{attribute 'linkalways'} 
{attribute 'no_explicit_call' := 'This FB is a CLASS and must be accessed using methods or properties'}
{attribute 'enable_dynamic_creation'}
FUNCTION_BLOCK _ETcVnColorTrainingMethod EXTENDS EnumDatatypeBase
VAR
	localData : ETcVnColorTrainingMethod;
	activeData : REFERENCE TO ETcVnColorTrainingMethod;
	enumBaseDatatype : _DINT(localData);
END_VAR

METHOD PRIVATE AddLocalEnumeration
VAR_INPUT
	Enumeration : T_MAXSTRING;
	Value : ETcVnColorTrainingMethod;
END_VAR
AddEnumeration(Enumeration, Value);
END_METHOD

PROPERTY PUBLIC Address : PVOID
GET
Address := ADR(activeData);
END_GET
END_PROPERTY

METHOD PUBLIC ClearReference
VAR_INPUT
END_VAR
activeData REF= localData;
SetBaseDatatypeReference();
END_METHOD

METHOD PUBLIC Clone : I_Datatype
VAR
    pClone : POINTER TO _ETcVnColorTrainingMethod;
END_VAR
pClone := __NEW(_ETcVnColorTrainingMethod(InitialValue := Value));
Clone := pClone^;
END_METHOD

METHOD FB_init : BOOL
VAR_INPUT
	bInitRetains : BOOL; // if TRUE, the retain variables are initialized (warm start / cold start)
	bInCopyCode : BOOL;  // if TRUE, the instance afterwards gets moved into the copy code (online change)
	InitialValue : ETcVnColorTrainingMethod;
END_VAR
localData := InitialValue;
AddBaseDatatype(enumBaseDatatype);
ClearReference();

AddLocalEnumeration('TCVN_CTM_LAB', ETcVnColorTrainingMethod.TCVN_CTM_LAB);
AddLocalEnumeration('TCVN_CTM_RGB', ETcVnColorTrainingMethod.TCVN_CTM_RGB);
END_METHOD

PROPERTY PUBLIC Identifier : T_MAXSTRING
GET
Identifier := 'ETcVnColorTrainingMethod';
END_GET
END_PROPERTY

METHOD IsEnumeratorValueEqual : BOOL
VAR_INPUT
	Enumerator : I_KeyValueForwardEnumerator;
END_VAR
VAR
	storedValue : ETcVnColorTrainingMethod;
END_VAR
IF NOT Enumerator.TryGet(storedValue) THEN
	RETURN;
END_IF

IsEnumeratorValueEqual := storedValue = activeData;
END_METHOD

METHOD PUBLIC MakeReferenceTo
VAR_INPUT
	ReferenceTarget : REFERENCE TO ETcVnColorTrainingMethod;
END_VAR
activeData REF= ReferenceTarget;
SetBaseDatatypeReference();
END_METHOD

METHOD PROTECTED SetBaseDatatypeReference
VAR_INPUT
END_VAR
enumBaseDatatype.MakeReferenceTo(activeData);
END_METHOD

PROPERTY PUBLIC Size : UDINT
GET
Size := SIZEOF(activeData);
END_GET
END_PROPERTY

METHOD TryMakeReferenceTo : BOOL
VAR_INPUT
	Target : I_Datatype;
END_VAR
VAR
	targetAsEnum : I_EnumDatatype;
	pTargetData : POINTER TO ETcVnColorTrainingMethod;
END_VAR
IF NOT Target.TryResolveAsEnumDatatype(targetAsEnum) THEN
	RETURN;
END_IF

IF targetAsEnum.Identifier <> Identifier THEN
	RETURN;
END_IF

pTargetData := Target.Address;
activeData REF= pTargetData^;
SetBaseDatatypeReference();
TryMakeReferenceTo := TRUE;
END_METHOD

PROPERTY PUBLIC Value : ETcVnColorTrainingMethod
GET
Value := activeData;
END_GET
SET
activeData := Value;
END_SET
END_PROPERTY

END_FUNCTION_BLOCK

(* stored: Version 1.1.0.1, ProductVersion 3.1.4024.12
   POU _ETcVnColorTrainingMethod: Id {6028da55-d8a0-0f8d-2afc-d94080e8e5ba}, SpecialFunc None
   Folder Constructor: Id {1bb38a8e-b814-0d41-3d43-d2efa85f6946}
   Folder Private: Id {cf11808f-3c76-0852-2ed6-f98f4ad7fced}
   Folder Protected: Id {f1175831-533e-03d6-3c3a-4faefcf5d79d}
   Method AddLocalEnumeration: Id {b7e3e48d-8aae-04b2-3d6c-7a977cbc5a40}
   Property Address: Id {b6820bd9-1f14-069c-2263-f363a84e71b0}
   Get Get: Id {9ad705a9-391b-01d9-0a6a-2dcb629bfc1d}
   Method ClearReference: Id {638f89f2-5d18-07f7-0871-123cb68304e9}
   Method Clone: Id {82db6a33-a5e5-01a1-14b1-9dd96bf7d688}
   Method FB_init: Id {3580fadd-f501-0afa-1fda-3530e26eb045}
   Property Identifier: Id {0f149496-b3d1-08c6-1eee-49ef345cf84e}
   Get Get: Id {7e3af238-043c-06ad-3e48-49416720f0da}
   Method IsEnumeratorValueEqual: Id {5e1dd4e3-1066-0fbe-2fc3-9e81e510c494}
   Method MakeReferenceTo: Id {ec6f9e4f-cdab-0f8f-384f-b11715e64901}
   Method SetBaseDatatypeReference: Id {766004f2-24a4-08f3-31b6-3a9b0f3660dd}
   Property Size: Id {9274ffc8-87b1-042e-1bfd-660f924cbf98}
   Get Get: Id {1877acff-e0a6-0ed3-2003-3ee55dcae07a}
   Method TryMakeReferenceTo: Id {fca9137e-2154-0a8f-03fc-1d221745d533}
   Property Value: Id {8f7584c3-8a8d-0ade-10d9-095454df7cdd}
   Get Get: Id {57e196b4-3379-0dc3-2640-ece7c13b52b5}
   Set Set: Id {9a680b1b-d3bc-0095-1b88-0b5d17e2f209} *)
